% RSLogix 500 project PROJECT9- DDE MEssaging.RSS, saved by version 8.30.00.16 %
PROJECT "UNTITLED"    % processor: Bul.1763 MicroLogix 1100 Series B %

PROGRAM FILES
  LAD 2   14 rungs

DATA FILES
  O0 OUTPUT  4 elements
  I1 INPUT  6 elements
  S2 STATUS  66 elements
  B3 BINARY  1 elements
  T4 TIMER  4 elements
  C5 COUNTER  1 elements
  R6 CONTROL  1 elements
  N7 INTEGER  10 elements
  F8 FLOAT  1 elements
  ST9 STRINGS  7 elements

LADDER 2
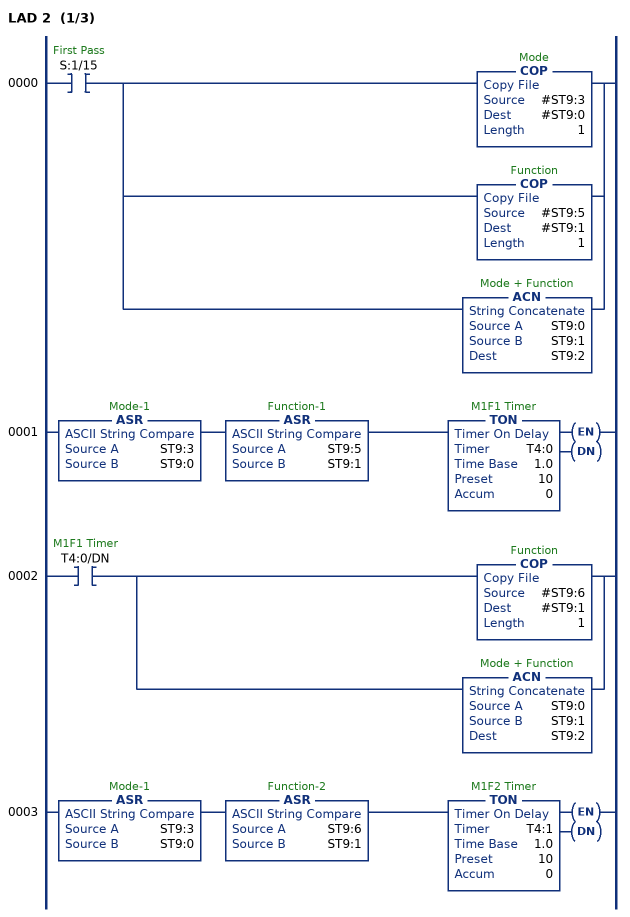
% Rung: 0 %
SOR XIC S:1/15 BST COP #ST9:3 #ST9:0 1 NXB COP #ST9:5 #ST9:1 1 NXB ACN ST9:0 ST9:1 ST9:2 BND EOR
%   S:1/15  "First Pass" %
%   ST9:3  "Mode-1" %
%   ST9:0  "Mode" %
%   ST9:5  "Function-1" %
%   ST9:1  "Function" %
%   ST9:2  "Mode + Function" %
% Rung: 1 %
SOR ASR ST9:3 ST9:0 ASR ST9:5 ST9:1 TON T4:0 1.0 10 0 EOR
%   ST9:3  "Mode-1" %
%   ST9:0  "Mode" %
%   ST9:5  "Function-1" %
%   ST9:1  "Function" %
%   T4:0  "M1F1 Timer" %
% Rung: 2 %
SOR XIC T4:0/DN BST COP #ST9:6 #ST9:1 1 NXB ACN ST9:0 ST9:1 ST9:2 BND EOR
%   T4:0  "M1F1 Timer" %
%   ST9:6  "Function-2" %
%   ST9:1  "Function" %
%   ST9:0  "Mode" %
%   ST9:2  "Mode + Function" %
% Rung: 3 %
SOR ASR ST9:3 ST9:0 ASR ST9:6 ST9:1 TON T4:1 1.0 10 0 EOR
%   ST9:3  "Mode-1" %
%   ST9:0  "Mode" %
%   ST9:6  "Function-2" %
%   ST9:1  "Function" %
%   T4:1  "M1F2 Timer" %

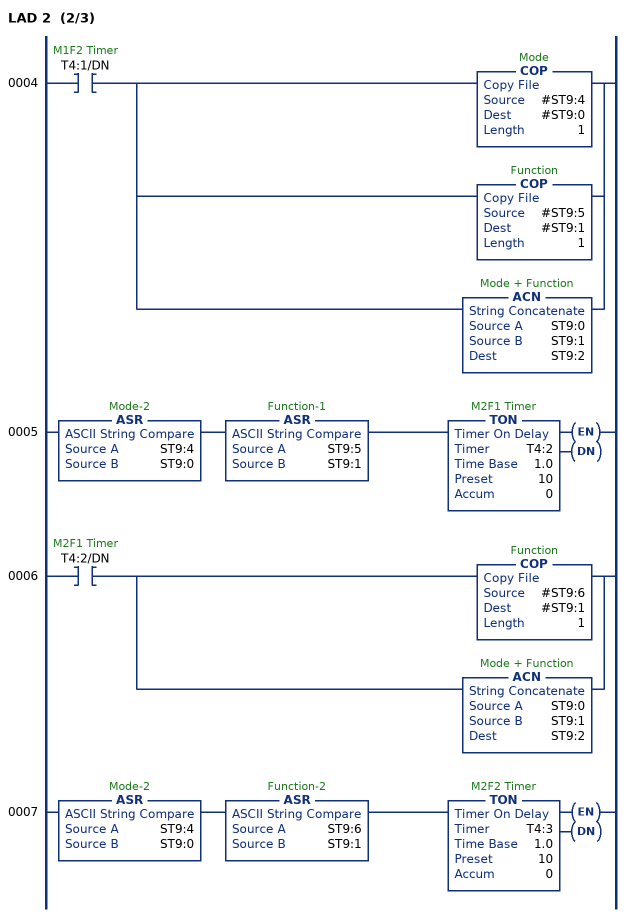
% Rung: 4 %
SOR XIC T4:1/DN BST COP #ST9:4 #ST9:0 1 NXB COP #ST9:5 #ST9:1 1 NXB ACN ST9:0 ST9:1 ST9:2 BND EOR
%   T4:1  "M1F2 Timer" %
%   ST9:4  "Mode-2" %
%   ST9:0  "Mode" %
%   ST9:5  "Function-1" %
%   ST9:1  "Function" %
%   ST9:2  "Mode + Function" %
% Rung: 5 %
SOR ASR ST9:4 ST9:0 ASR ST9:5 ST9:1 TON T4:2 1.0 10 0 EOR
%   ST9:4  "Mode-2" %
%   ST9:0  "Mode" %
%   ST9:5  "Function-1" %
%   ST9:1  "Function" %
%   T4:2  "M2F1 Timer" %
% Rung: 6 %
SOR XIC T4:2/DN BST COP #ST9:6 #ST9:1 1 NXB ACN ST9:0 ST9:1 ST9:2 BND EOR
%   T4:2  "M2F1 Timer" %
%   ST9:6  "Function-2" %
%   ST9:1  "Function" %
%   ST9:0  "Mode" %
%   ST9:2  "Mode + Function" %
% Rung: 7 %
SOR ASR ST9:4 ST9:0 ASR ST9:6 ST9:1 TON T4:3 1.0 10 0 EOR
%   ST9:4  "Mode-2" %
%   ST9:0  "Mode" %
%   ST9:6  "Function-2" %
%   ST9:1  "Function" %
%   T4:3  "M2F2 Timer" %

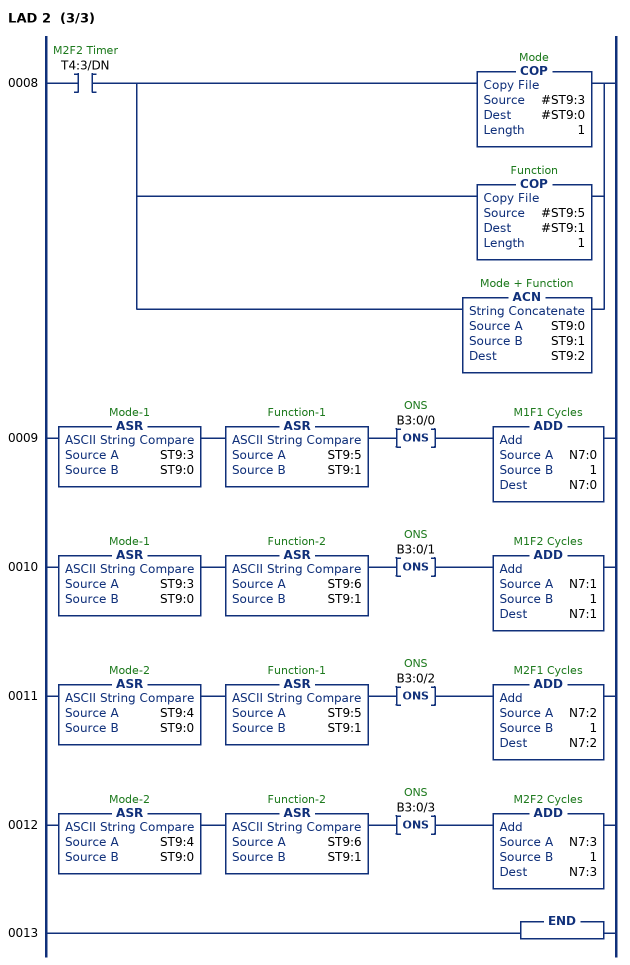
% Rung: 8 %
SOR XIC T4:3/DN BST COP #ST9:3 #ST9:0 1 NXB COP #ST9:5 #ST9:1 1 NXB ACN ST9:0 ST9:1 ST9:2 BND EOR
%   T4:3  "M2F2 Timer" %
%   ST9:3  "Mode-1" %
%   ST9:0  "Mode" %
%   ST9:5  "Function-1" %
%   ST9:1  "Function" %
%   ST9:2  "Mode + Function" %
% Rung: 9 %
SOR ASR ST9:3 ST9:0 ASR ST9:5 ST9:1 ONS B3:0/0 ADD N7:0 1 N7:0 EOR
%   ST9:3  "Mode-1" %
%   ST9:0  "Mode" %
%   ST9:5  "Function-1" %
%   ST9:1  "Function" %
%   B3:0/0  "ONS" %
%   N7:0  "M1F1 Cycles" %
% Rung: 10 %
SOR ASR ST9:3 ST9:0 ASR ST9:6 ST9:1 ONS B3:0/1 ADD N7:1 1 N7:1 EOR
%   ST9:3  "Mode-1" %
%   ST9:0  "Mode" %
%   ST9:6  "Function-2" %
%   ST9:1  "Function" %
%   B3:0/1  "ONS" %
%   N7:1  "M1F2 Cycles" %
% Rung: 11 %
SOR ASR ST9:4 ST9:0 ASR ST9:5 ST9:1 ONS B3:0/2 ADD N7:2 1 N7:2 EOR
%   ST9:4  "Mode-2" %
%   ST9:0  "Mode" %
%   ST9:5  "Function-1" %
%   ST9:1  "Function" %
%   B3:0/2  "ONS" %
%   N7:2  "M2F1 Cycles" %
% Rung: 12 %
SOR ASR ST9:4 ST9:0 ASR ST9:6 ST9:1 ONS B3:0/3 ADD N7:3 1 N7:3 EOR
%   ST9:4  "Mode-2" %
%   ST9:0  "Mode" %
%   ST9:6  "Function-2" %
%   ST9:1  "Function" %
%   B3:0/3  "ONS" %
%   N7:3  "M2F2 Cycles" %
% Rung: 13 %
SOR END EOR

DATA TABLE (non-zero values as saved)
DATA T4
% .PRE .ACC %
% T4:0 % 10 0
% T4:1 % 10 0
% T4:2 % 10 0
% T4:3 % 10 0
DATA ST9
% ST9:3 % "Mode-1"
% ST9:4 % "Mode-2"
% ST9:5 % "F1"
% ST9:6 % "F2"
